INTERFACE ITF_TopElement1_HMI_Connector_View EXTENDS ITF_BaseTopElement_HMI_Connector_View

END_INTERFACE

(* stored: Version 1.1.0.1
   Itf ITF_TopElement1_HMI_Connector_View: Id {e9c1d5b7-68a8-0560-18e3-bd57adcda597} *)
